(*
SPDX-FileCopyrightText: © 2026 Oleksandr Tiutyk <trofimich@gmail.com>
SPDX-License-Identifier: MIT
License: https://opensource.org/license/mit
*)

(*!
<summary>
Beckhoff EL1018: 8-channel fast digital input terminal (24 V DC, 10 µs filter).
</summary>
<description>
Process image mapping structure for the EL1018 fast EtherCAT terminal with 8 discrete 24 V DC inputs and 10
µs input filter.
When used for I/O, link located fields or their containing buffers to the matching selected PDOs.
The record is not a packed wire buffer; compiler padding is not part of the device specification.
Unlinked/default values do not prove valid I/O. The caller evaluates bus/channel validity before use.
Use one owner task per instance and externally synchronize other access; multi-field snapshots are not atomic.
Copies store data without creating hardware links. Keep borrowed field references valid while consumers are bound.
This passive record performs no validation, synchronization, configuration or protocol advancement.
</description>
*)
TYPE EL1018 :
STRUCT
	Ch1 AT %I* : BOOL;
	Ch2 AT %I* : BOOL;
	Ch3 AT %I* : BOOL;
	Ch4 AT %I* : BOOL;
	Ch5 AT %I* : BOOL;
	Ch6 AT %I* : BOOL;
	Ch7 AT %I* : BOOL;
	Ch8 AT %I* : BOOL;
END_STRUCT
END_TYPE

(* stored: Version 1.1.0.1, ProductVersion 3.1.4026.20
   DUT EL1018: Id {5869f5ee-46b2-4f87-9be4-4310329fae1d} *)
